# B&R Automation Studio project Ironer_Line
Automation Studio 4.4.4.112; technology packages: mappView 5.1.1

## Configuration Config1

### IoMap.iom - X20CP0484/IoMap.iom
```iecst
VAR_CONFIG
	::T_tank AT %IW."X20AT4222-1".Temperature01;
	::inverter.CTRL_set AT %QW."8I66xxxxxxx.0P-xxx".CMDD_Output;
	::inverter.RPM_set AT %QW."8I66xxxxxxx.0P-xxx".LFRD_Output;
	::inverter.RPM_actual AT %IW."8I66xxxxxxx.0P-xxx".RFRD_Input;
	::inverter.freq AT %IW."8I66xxxxxxx.0P-xxx".RFR_Input;
	::inverter.voltage AT %IW."8I66xxxxxxx.0P-xxx".UOP_Input;
	::inverter.current AT %IW."8I66xxxxxxx.0P-xxx".LCR_Input;
	::inverter.DC AT %IW."8I66xxxxxxx.0P-xxx".ULN_Input;
	::inverter.error_code AT %IW."8I66xxxxxxx.0P-xxx".ERRD_Input;
	::inverter.CTRL_actual AT %IW."8I66xxxxxxx.0P-xxx".ETAD_Input;
	::inverter.RPM_after_ramp AT %IW."8I66xxxxxxx.0P-xxx".FROD_Input;
	::mulde_3.T_out AT %IW."X20AT4222-4".Temperature02;
	::mulde_3.T_in AT %IW."X20AT4222-4".Temperature01;
	::mulde_1.T_in AT %IW."X20AT4222-2".Temperature01;
	::mulde_2.T_out AT %IW."X20AT4222-3".Temperature02;
	::mulde_2.T_in AT %IW."X20AT4222-3".Temperature01;
	::mulde_1.T_out AT %IW."X20AT4222-2".Temperature02;
	::heater AT %QX."X20DO9322".DigitalOutput01;
END_VAR
```

## Logical view

Binary libraries used (declarations not repeated): operator, runtime, astime, AsIecCon

### Global.typ - Global data types
```iecst
TYPE
	Inverter_type : 	STRUCT
		CTRL_Word : UINT;
		Set_RPM : INT;
		Actual_CTRL_Word : UINT;
		RPM_After_Ramp : INT;
		Error_Code : UINT;
		DC : UINT;
		Voltage : UINT;
		Current : UINT;
		Actual_Out_fq : INT;
		Actual_RMP : INT;
	END_STRUCT;
END_TYPE
```

### Global.var - Global variables
```iecst
VAR
	mulde_3 : mulde_type;
	mulde_2 : mulde_type;
	mulde_1 : mulde_type;
	inverter : inverter_type;
	p_pumpe : p_pumpe_type;
	T_tank : INT;
	heater : BOOL;
	p_last : USINT;
END_VAR
```

### Package Logical/Libraries - Global libraries

- Visualisation Logical/mappView (not shown)

Listed in the project but not available here: Logical/Program
